(* PLC project SafeLOGIC-1, BrAutomation SafeDESIGNER  4.2.0.17 *)
(* stored: companyURL http://www.br-automation.com, creationDateTime Thu Nov 03 12:56:04 2016 *)

PROGRAM Main
  VAR  (* added by the conversion: wires and edge detectors of the diagram *)
    _AND_S53_OUT : ANY;
  END_VAR

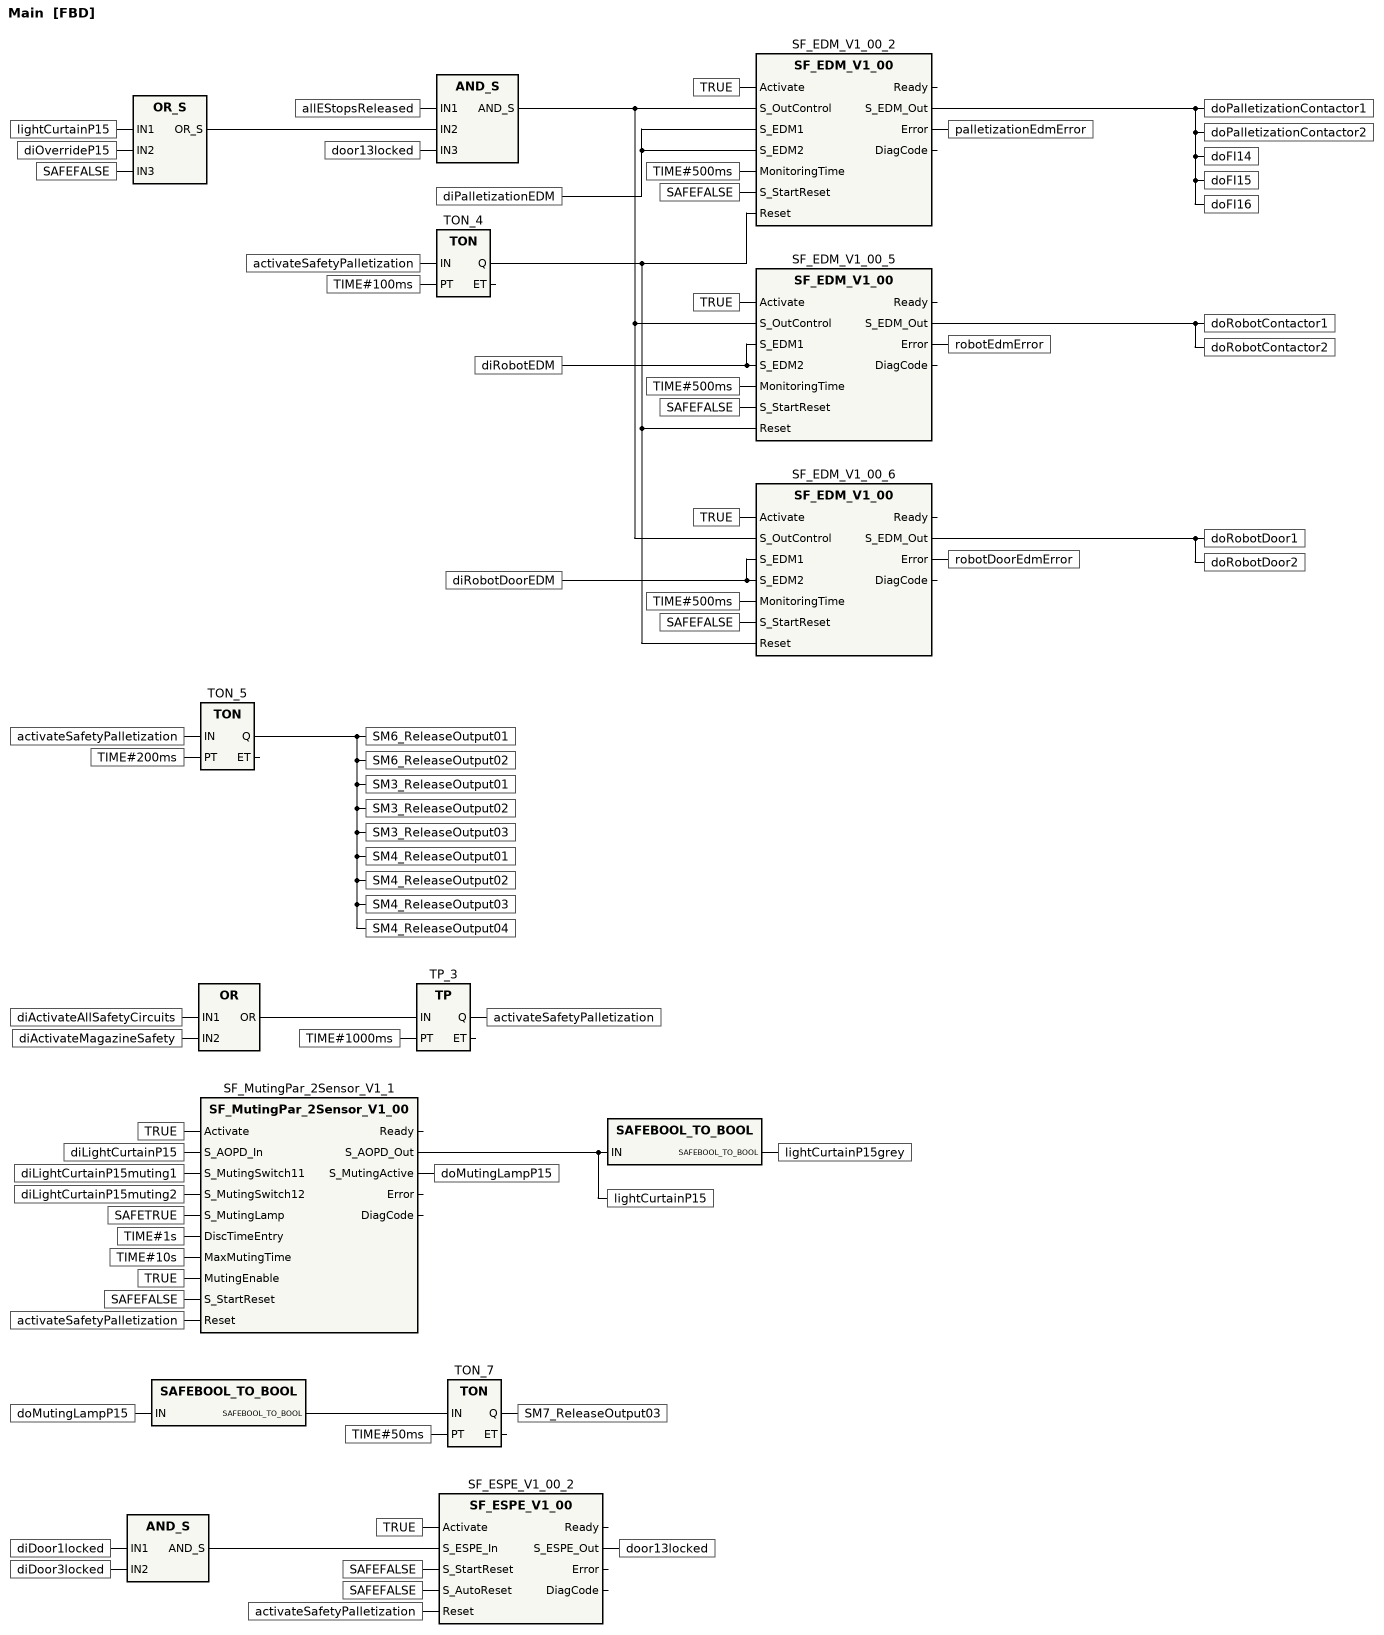
(* FBD diagram, written out as Structured Text *)
TP_3(IN := diActivateAllSafetyCircuits OR diActivateMagazineSafety, PT := TIME#1000ms);
activateSafetyPalletization := TP_3.Q;
SF_MutingPar_2Sensor_V1_1(Activate := TRUE, S_AOPD_In := diLightCurtainP15, S_MutingSwitch11 := diLightCurtainP15muting1, S_MutingSwitch12 := diLightCurtainP15muting2, S_MutingLamp := SAFETRUE, DiscTimeEntry := TIME#1s, MaxMutingTime := TIME#10s, MutingEnable := TRUE, S_StartReset := SAFEFALSE, Reset := activateSafetyPalletization);
doMutingLampP15 := SF_MutingPar_2Sensor_V1_1.S_MutingActive;
lightCurtainP15 := SF_MutingPar_2Sensor_V1_1.S_AOPD_Out;
lightCurtainP15grey := SAFEBOOL_TO_BOOL(SF_MutingPar_2Sensor_V1_1.S_AOPD_Out);
SF_ESPE_V1_00_2(Activate := TRUE, S_ESPE_In := AND_S(diDoor1locked, diDoor3locked), S_StartReset := SAFEFALSE, S_AutoReset := SAFEFALSE, Reset := activateSafetyPalletization);
door13locked := SF_ESPE_V1_00_2.S_ESPE_Out;
_AND_S53_OUT := AND_S(allEStopsReleased, OR_S(lightCurtainP15, diOverrideP15, SAFEFALSE), door13locked);
TON_4(IN := activateSafetyPalletization, PT := TIME#100ms);
SF_EDM_V1_00_2(Activate := TRUE, S_OutControl := _AND_S53_OUT, S_EDM1 := diPalletizationEDM, S_EDM2 := diPalletizationEDM, MonitoringTime := TIME#500ms, S_StartReset := SAFEFALSE, Reset := TON_4.Q);
palletizationEdmError := SF_EDM_V1_00_2.Error;
doPalletizationContactor1 := SF_EDM_V1_00_2.S_EDM_Out;
doPalletizationContactor2 := SF_EDM_V1_00_2.S_EDM_Out;
doFI15 := SF_EDM_V1_00_2.S_EDM_Out;
doFI14 := SF_EDM_V1_00_2.S_EDM_Out;
doFI16 := SF_EDM_V1_00_2.S_EDM_Out;
SF_EDM_V1_00_5(Activate := TRUE, S_OutControl := _AND_S53_OUT, S_EDM1 := diRobotEDM, S_EDM2 := diRobotEDM, MonitoringTime := TIME#500ms, S_StartReset := SAFEFALSE, Reset := TON_4.Q);
robotEdmError := SF_EDM_V1_00_5.Error;
doRobotContactor1 := SF_EDM_V1_00_5.S_EDM_Out;
doRobotContactor2 := SF_EDM_V1_00_5.S_EDM_Out;
SF_EDM_V1_00_6(Activate := TRUE, S_OutControl := _AND_S53_OUT, S_EDM1 := diRobotDoorEDM, S_EDM2 := diRobotDoorEDM, MonitoringTime := TIME#500ms, S_StartReset := SAFEFALSE, Reset := TON_4.Q);
robotDoorEdmError := SF_EDM_V1_00_6.Error;
doRobotDoor1 := SF_EDM_V1_00_6.S_EDM_Out;
doRobotDoor2 := SF_EDM_V1_00_6.S_EDM_Out;
TON_5(IN := activateSafetyPalletization, PT := TIME#200ms);
SM6_ReleaseOutput02 := TON_5.Q;
SM6_ReleaseOutput01 := TON_5.Q;
SM3_ReleaseOutput01 := TON_5.Q;
SM3_ReleaseOutput02 := TON_5.Q;
SM3_ReleaseOutput03 := TON_5.Q;
SM4_ReleaseOutput02 := TON_5.Q;
SM4_ReleaseOutput01 := TON_5.Q;
SM4_ReleaseOutput03 := TON_5.Q;
SM4_ReleaseOutput04 := TON_5.Q;
TON_7(IN := SAFEBOOL_TO_BOOL(doMutingLampP15), PT := TIME#50ms);
SM7_ReleaseOutput03 := TON_7.Q;
END_PROGRAM
